{attribute 'Tc2GvlVarNames'}
VAR_CONFIG
END_VAR

(* stored: Version 1.1.0.1, ProductVersion 3.1.4024.6
   GVL Variable_Configuration: Id {029be460-4d18-4e71-b323-5df0a572faf9} *)
